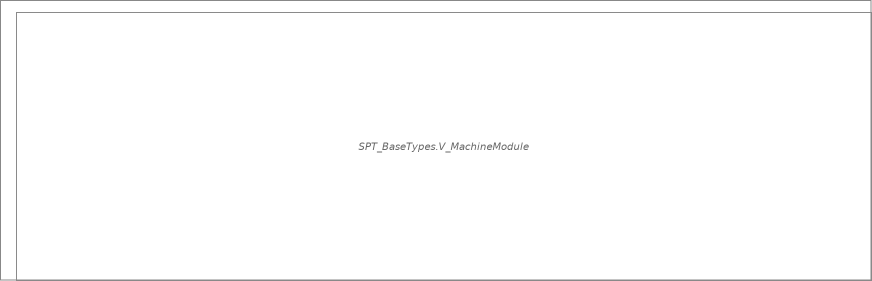
VISUALIZATION Visualization  // 872x281
    Frame (16,12 856x269)
        shows SPT_BaseTypes.V_MachineModule(HMI := MAIN.Machine.PackMLBaseModule_HMI)
END_VISUALIZATION

(* stored: Version 1.1.0.1, ProductVersion 3.1.4026.12
   Visu Visualization: Id {f15c2a30-041d-4b7a-b80a-8fc5d0c26b64} *)
